(* IEC 61131-3 sources: test/Class/pumpControl, 1 file *)

(* ---- pumpControl.st ---- *)
#define test 1

(*!
<Class
	Name               = "pumpControl"
	Revision           = "0.0"
	RealtimeTask       = "false"
	CyclicTask         = "true"
	DefCyclictime      = "10 ms"
	BackgroundTask     = "false"
	Sigmatek           = "false"
	OSInterface        = "false"
	HighPriority       = "false"
	Automatic          = "false"
	UpdateMode         = "Prescan"
	SharedCommandTable = "true"
	Objectsize         = "(484,120)">
	<Channels>
		<Server Name="ActFillLevelVisu" Visualized="true" Initialize="false" WriteProtected="true" Retentive="false"/>
		<Server Name="ClassSvr" Visualized="false" Initialize="false" WriteProtected="true" Retentive="false"/>
		<Server Name="MaxBorder" Visualized="true" Initialize="true" DefValue="800" WriteProtected="false" Retentive="File"/>
		<Server Name="MinBorder" Visualized="true" Initialize="false" WriteProtected="false" Retentive="File"/>
		<Server Name="PumpVisu" Visualized="true" Initialize="false" WriteProtected="true" Retentive="false"/>
		<Server Name="tt" Visualized="true" Initialize="false" WriteProtected="true" Retentive="false"/>
		<Server Name="ttt" Visualized="true" Initialize="false" WriteProtected="true" Retentive="false"/>
		<Server Name="tttt" Visualized="true" Initialize="false" WriteProtected="true" Retentive="false"/>
		<Client Name="ActFillLevel" Required="false" Internal="false"/>
		<Client Name="Pump" Required="false" Internal="false"/>
		<Client Name="test1" Required="false" Internal="false"/>
		<Client Name="test2" Required="false" Internal="false"/>
	</Channels>
</Class>
*)
pumpControl : CLASS
  //Servers:
	ClassSvr 	: SvrChCmd_DINT;
	MaxBorder 	: SvrCh_DINT;
	MinBorder 	: SvrCh_DINT;
	ActFillLevelVisu 	: SvrCh_DINT;
	PumpVisu 	: SvrCh_DINT;
	tt 	: SvrCh_DINT;
	ttt 	: SvrCh_DINT;
	tttt 	: SvrCh_DINT;
  //Clients:
	Pump 	: CltCh_DINT;
	ActFillLevel 	: CltCh_DINT;
	test2 	: CltCh_DINT;
	test1 	: CltCh_DINT;
  //Variables:
		pu 	: DINT;
  //Functions:

	FUNCTION VIRTUAL GLOBAL CyWork
		VAR_INPUT
			EAX 	: UDINT;
		END_VAR
		VAR_OUTPUT
			state (EAX) 	: UDINT;
		END_VAR;

	FUNCTION VIRTUAL GLOBAL ActFillLevelVisu::Read
		VAR_OUTPUT
			output (EAX) 	: DINT;
		END_VAR;

	FUNCTION VIRTUAL GLOBAL PumpVisu::Read
		VAR_OUTPUT
			output (EAX) 	: DINT;
		END_VAR;
  //Tables:
	FUNCTION @STD
		VAR_OUTPUT
			ret_code	: CONFSTATES;
		END_VAR;
	FUNCTION GLOBAL TAB @CT_;
END_CLASS;

FUNCTION VIRTUAL GLOBAL pumpControl::CyWork
	VAR_INPUT
		EAX 	: UDINT;
	END_VAR
	VAR_OUTPUT
		state (EAX) 	: UDINT;
	END_VAR
  ActFillLevel := ActFillLevel.Read();
  pu := ActFillLevel;
  if ActFillLevel >= MaxBorder then
    pump := 1;
  elsif ActFillLevel <= MinBorder then
    pump := 0;
  end_if;

  Pump.Write (Pump);
	state := READY;

END_FUNCTION

FUNCTION VIRTUAL GLOBAL pumpControl::ActFillLevelVisu::Read
	VAR_OUTPUT
		output (EAX) 	: DINT;
	END_VAR

	ActFillLevelVisu := ActFillLevel;

	output := ActFillLevelVisu;

END_FUNCTION

FUNCTION VIRTUAL GLOBAL pumpControl::PumpVisu::Read
	VAR_OUTPUT
		output (EAX) 	: DINT;
	END_VAR

	PumpVisu := Pump;

	output := PumpVisu;

END_FUNCTION
